// TIA Portal V20 export
DATA_BLOCK "Main_Safety_RTG1_DB"   // DB6, F_DB
NAME : FUSI
// stored: InstanceOfName Main_Safety_RTG1, InstanceOfType FB
"Main_Safety_RTG1"
   // VAR
   //    ESTOP1 : ESTOP1;
   // END_VAR
BEGIN
END_DATA_BLOCK
